// TIA Portal V20 export
TYPE "s_CONNECTION_STATUS"
// stored: Access Published, IsFailsafeCompliant true, Namespace Safety
   STRUCT
      RunMode { ExternalWritable := 'False'} : Bool := FALSE;   // station is running on automode
      ConnectionFault { ExternalWritable := 'False'} : Bool := FALSE;   // communication fault on F-link
   END_STRUCT;
END_TYPE
